Yaskawa INFORM job: L_F_BOTTOM_S2.JBI

/JOB
//NAME L_F_BOTTOM_S2
//POS
///NPOS 10,10,10,0,0,0
///TOOL 2
///POSTYPE PULSE
///PULSE
C00000=-121870,88665,73064,21827,-2155,-30652
C00001=-121988,80124,46976,22117,8778,-32513
C00002=-122013,79915,42787,22335,11015,-32906
C00003=-122023,79968,41268,22435,11878,-33060
C00004=-122061,74540,35092,22584,13044,-33263
C00005=-122177,59887,19029,23012,15853,-33760
C00006=-122217,55364,14259,23147,16615,-33896
C00007=-122206,54996,15466,23003,15797,-33741
C00008=-122179,54316,18722,22676,13716,-33355
C00009=-122069,55578,35868,21862,4730,-31782
///TOOL 0
BC00000=223981
BC00001=223981
BC00002=223981
BC00003=223981
BC00004=224001
BC00005=224062
BC00006=224082
BC00007=224082
BC00008=224082
BC00009=224082
EC00000=-568526,175863
EC00001=-568526,175863
EC00002=-568526,175863
EC00003=-568526,175863
EC00004=-568526,175863
EC00005=-568526,175863
EC00006=-568526,175863
EC00007=-568526,175863
EC00008=-568526,175863
EC00009=-568526,175863
//INST
///DATE 2026/05/13 10:02
///ATTR SC,RW
///GROUP1 RB1,BS1
///GROUP2 ST1
NOP
'L_F_bottom_s2
MEMOF
CLEAR MPF
'Path W2
SSFTOF
MOVJ C00000 BC00000 VJ=100.00  +MOVJ EC00000 VJ=100.00
SMOVL C00001 BC00001 V=1000.0  +MOVJ EC00001
SMOVL C00002 BC00002 V=400.0  +MOVJ EC00002
SMOVL C00003 BC00003 V=10.0 PL=0  +MOVJ EC00003
SMOVL C00004 BC00004 V=10.0  +MOVJ EC00004
SMOVL C00005 BC00005 V=10.0  +MOVJ EC00005
SMOVL C00006 BC00006 V=10.0  +MOVJ EC00006
SMOVL C00007 BC00007 V=400.0  +MOVJ EC00007
SMOVL C00008 BC00008 V=1000.0  +MOVJ EC00008
SMOVL C00009 BC00009 V=1000.0  +MOVJ EC00009
'EndPath W2
END
